PROGRAM MAIN
VAR_INPUT
END_VAR
VAR_OUTPUT
END_VAR
VAR
	Pump01						: PumpControl;
	ManAutoPb					: BOOL;
	ManPumpStart				: BOOL;						// N.O.
	ManPumpStop					: BOOL := TRUE;				// N.C.
	LevelSensorMin				: BOOL := TRUE;				// N.C.
	LevelSensorMax				: BOOL := TRUE;				// N.C.
	PumpRunning					: BOOL;
	ManAutoState				: BOOL;
END_VAR

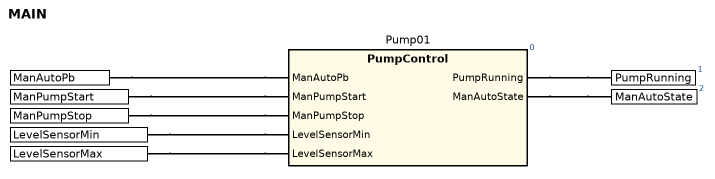
Pump01(
    ManAutoPb := ManAutoPb,
    ManPumpStart := ManPumpStart,
    ManPumpStop := ManPumpStop,
    LevelSensorMin := LevelSensorMin,
    LevelSensorMax := LevelSensorMax); // PumpControl
PumpRunning := Pump01.PumpRunning;
ManAutoState := Pump01.ManAutoState;

END_PROGRAM

(* stored: Version 1.1.0.1, ProductVersion 3.1.4024.15
   POU MAIN: Id {7aa3ffe1-ebb8-4c13-828a-c6b6b2732967}, SpecialFunc None *)
